{attribute 'qualified_only'}
VAR_GLOBAL
END_VAR

(* stored: Version 1.1.0.1, ProductVersion 3.1.4024.2
   GVL GVL: Id {3b6372bb-3e25-4d24-93d5-b62adc93e406} *)
